PROGRAM SP1_1_Y110
VAR
	CompareOutput110_00: CMP_OC_DW;
	CompareOutput110_01: CMP_OC_DW;
	CompareOutput110_02: CMP_OC_DW;
	CompareOutput110_03: CMP_OC_DW;
	CompareOutput110_04: CMP_OC_DW;
	CompareOutput110_05: CMP_OC_DW;
	CompareOutput110_06: CMP_OC_DW;
	CompareOutput110_07: CMP_OC_DW;
	CompareOutput110_08: CMP_OC_DW;
	CompareOutput110_09: CMP_OC_DW;
	CompareOutput110_10: CMP_OC_DW;
	CompareOutput110_11: CMP_OC_DW;
	CompareOutput110_12: CMP_OC_DW;
	CompareOutput110_13: CMP_OC_DW;
	CompareOutput110_14: CMP_OC_DW;
	CompareOutput110_15: CMP_OC_DW;

END_VAR

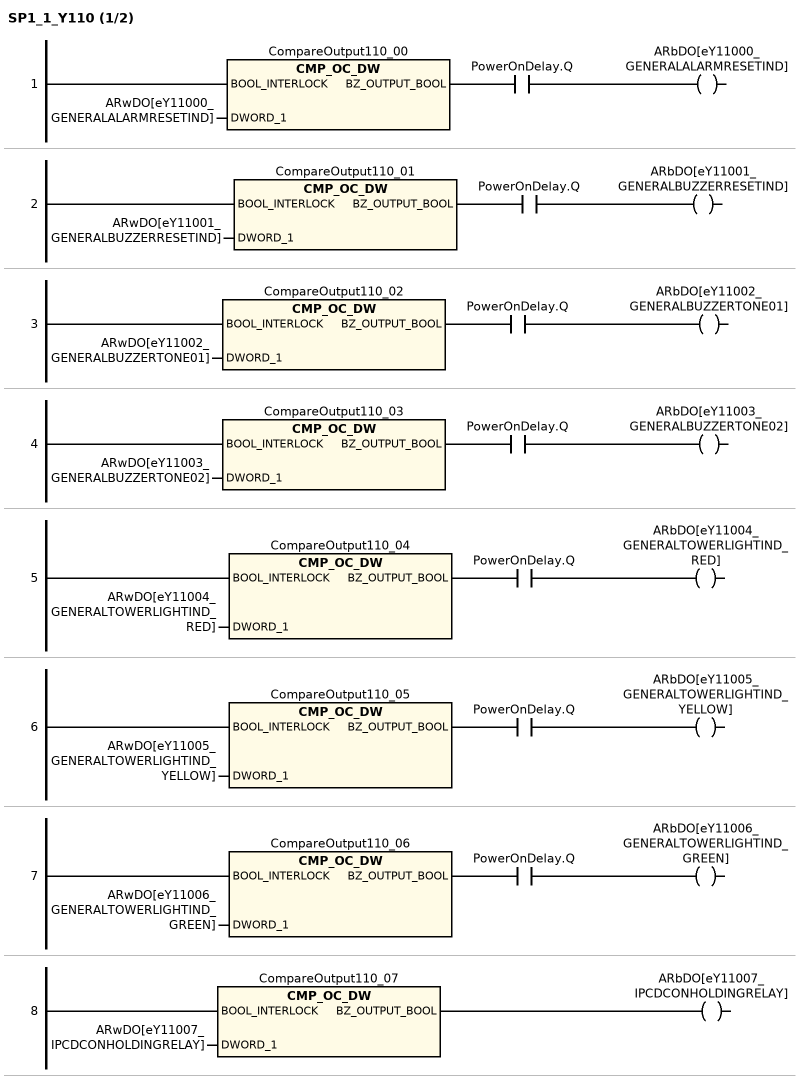
// NETWORK 1
CompareOutput110_00(BOOL_INTERLOCK := TRUE, DWORD_1 := ARwDO[eY11000_GENERALALARMRESETIND]); // CMP_OC_DW
ARbDO[eY11000_GENERALALARMRESETIND] := CompareOutput110_00.BZ_OUTPUT_BOOL AND PowerOnDelay.Q;

// NETWORK 2
CompareOutput110_01(BOOL_INTERLOCK := TRUE, DWORD_1 := ARwDO[eY11001_GENERALBUZZERRESETIND]); // CMP_OC_DW
ARbDO[eY11001_GENERALBUZZERRESETIND] := CompareOutput110_01.BZ_OUTPUT_BOOL AND PowerOnDelay.Q;

// NETWORK 3
CompareOutput110_02(BOOL_INTERLOCK := TRUE, DWORD_1 := ARwDO[eY11002_GENERALBUZZERTONE01]); // CMP_OC_DW
ARbDO[eY11002_GENERALBUZZERTONE01] := CompareOutput110_02.BZ_OUTPUT_BOOL AND PowerOnDelay.Q;

// NETWORK 4
CompareOutput110_03(BOOL_INTERLOCK := TRUE, DWORD_1 := ARwDO[eY11003_GENERALBUZZERTONE02]); // CMP_OC_DW
ARbDO[eY11003_GENERALBUZZERTONE02] := CompareOutput110_03.BZ_OUTPUT_BOOL AND PowerOnDelay.Q;

// NETWORK 5
CompareOutput110_04(BOOL_INTERLOCK := TRUE, DWORD_1 := ARwDO[eY11004_GENERALTOWERLIGHTIND_RED]); // CMP_OC_DW
ARbDO[eY11004_GENERALTOWERLIGHTIND_RED] := CompareOutput110_04.BZ_OUTPUT_BOOL AND PowerOnDelay.Q;

// NETWORK 6
CompareOutput110_05(BOOL_INTERLOCK := TRUE, DWORD_1 := ARwDO[eY11005_GENERALTOWERLIGHTIND_YELLOW]); // CMP_OC_DW
ARbDO[eY11005_GENERALTOWERLIGHTIND_YELLOW] := CompareOutput110_05.BZ_OUTPUT_BOOL AND PowerOnDelay.Q;

// NETWORK 7
CompareOutput110_06(BOOL_INTERLOCK := TRUE, DWORD_1 := ARwDO[eY11006_GENERALTOWERLIGHTIND_GREEN]); // CMP_OC_DW
ARbDO[eY11006_GENERALTOWERLIGHTIND_GREEN] := CompareOutput110_06.BZ_OUTPUT_BOOL AND PowerOnDelay.Q;

// NETWORK 8
CompareOutput110_07(BOOL_INTERLOCK := TRUE, DWORD_1 := ARwDO[eY11007_IPCDCONHOLDINGRELAY]); // CMP_OC_DW
ARbDO[eY11007_IPCDCONHOLDINGRELAY] := CompareOutput110_07.BZ_OUTPUT_BOOL;

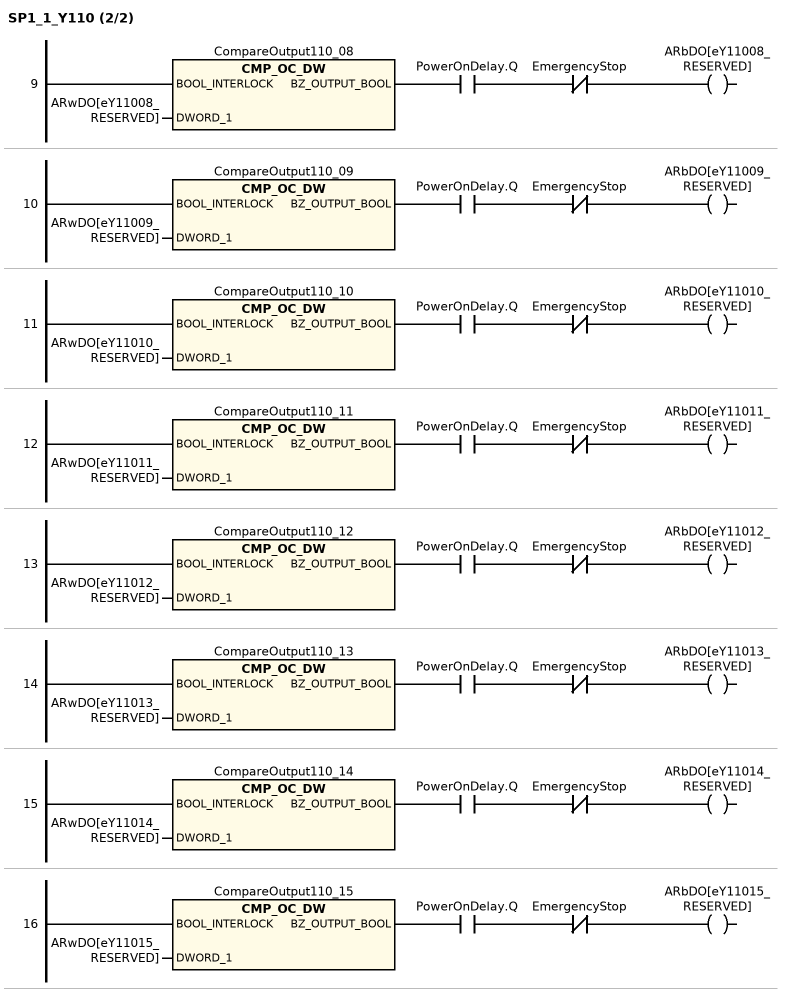
// NETWORK 9
CompareOutput110_08(BOOL_INTERLOCK := TRUE, DWORD_1 := ARwDO[eY11008_RESERVED]); // CMP_OC_DW
ARbDO[eY11008_RESERVED] := CompareOutput110_08.BZ_OUTPUT_BOOL AND PowerOnDelay.Q AND NOT EmergencyStop;

// NETWORK 10
CompareOutput110_09(BOOL_INTERLOCK := TRUE, DWORD_1 := ARwDO[eY11009_RESERVED]); // CMP_OC_DW
ARbDO[eY11009_RESERVED] := CompareOutput110_09.BZ_OUTPUT_BOOL AND PowerOnDelay.Q AND NOT EmergencyStop;

// NETWORK 11
CompareOutput110_10(BOOL_INTERLOCK := TRUE, DWORD_1 := ARwDO[eY11010_RESERVED]); // CMP_OC_DW
ARbDO[eY11010_RESERVED] := CompareOutput110_10.BZ_OUTPUT_BOOL AND PowerOnDelay.Q AND NOT EmergencyStop;

// NETWORK 12
CompareOutput110_11(BOOL_INTERLOCK := TRUE, DWORD_1 := ARwDO[eY11011_RESERVED]); // CMP_OC_DW
ARbDO[eY11011_RESERVED] := CompareOutput110_11.BZ_OUTPUT_BOOL AND PowerOnDelay.Q AND NOT EmergencyStop;

// NETWORK 13
CompareOutput110_12(BOOL_INTERLOCK := TRUE, DWORD_1 := ARwDO[eY11012_RESERVED]); // CMP_OC_DW
ARbDO[eY11012_RESERVED] := CompareOutput110_12.BZ_OUTPUT_BOOL AND PowerOnDelay.Q AND NOT EmergencyStop;

// NETWORK 14
CompareOutput110_13(BOOL_INTERLOCK := TRUE, DWORD_1 := ARwDO[eY11013_RESERVED]); // CMP_OC_DW
ARbDO[eY11013_RESERVED] := CompareOutput110_13.BZ_OUTPUT_BOOL AND PowerOnDelay.Q AND NOT EmergencyStop;

// NETWORK 15
CompareOutput110_14(BOOL_INTERLOCK := TRUE, DWORD_1 := ARwDO[eY11014_RESERVED]); // CMP_OC_DW
ARbDO[eY11014_RESERVED] := CompareOutput110_14.BZ_OUTPUT_BOOL AND PowerOnDelay.Q AND NOT EmergencyStop;

// NETWORK 16
CompareOutput110_15(BOOL_INTERLOCK := TRUE, DWORD_1 := ARwDO[eY11015_RESERVED]); // CMP_OC_DW
ARbDO[eY11015_RESERVED] := CompareOutput110_15.BZ_OUTPUT_BOOL AND PowerOnDelay.Q AND NOT EmergencyStop;

END_PROGRAM

(* stored: Version 1.1.0.1, ProductVersion 3.1.4024.11
   POU SP1_1_Y110: Id {d320ed5d-c316-41a6-96a0-aa1a4422b697}, SpecialFunc None *)
